TYPE ST_M001_Interface :
STRUCT
	bRunCycle,
	bEmptyPlant : BOOL;
END_STRUCT
END_TYPE

(* stored: Version 1.1.0.1
   DUT ST_M001_Interface: Id {7a95c9fb-c0b7-4d72-b6d6-fa0bcabbfcb4} *)
